(* CoDeSys 2.3.8.1 project: House.pro *)
(* Libraries: Standard.lib 4.10.05 12:14:46, IecSfc.lib 13.4.06 16:51:28, SYSLIBCALLBACK.LIB 16.4.07 17:52:46 *)

(* Global variable list: Global_Variables *)
VAR_GLOBAL
	(* Контроль 0 *)
	G_IN_CTL_BTN_1: BOOL; (* Кнопка ALL *)
	G_IN_CTL_BTN_2: BOOL; (* Кнопка RESET *)
	G_OUT_CTL_ALARM_LAMP: BOOL; (* Лампа-сигнализатор *)
	G_OUT_CTL_ALARM_SOUND: BOOL; (* Динамик в ПЛК *)
	G_OUT_CTL_SOCKET_1: BOOL := TRUE; (* Питание для МВВ *)

	(* Дверь *)
	G_IN_DOOR_DTR_1: BOOL; (* Сенсор открытия двери *)
	G_IN_DOOR_BTN_BELL: BOOL; (* Кнопка звонка *)
	G_OUT_DOOR_BELL: BOOL; (* Звонок *)

	(* Кухня 1 *)
	G_IN_KTN_BTN_1: BOOL; (* Выключатель основной *)
	G_IN_KTN_BTN_2: BOOL; (* Выключатель для вытяжки *)
	G_IN_KTN_DTR_1: BOOL; (* Датчик протечек *)
	G_OUT_KTN_LIGHT_1: BOOL; (* Свет основной *)
	G_OUT_KTN_LIGHT_2: BOOL; (* Свет второстепенный (подсветка) *)
	G_OUT_KTN_FAN_1: BOOL; (* Вытяжка *)

	(* Балкон *)
	G_IN_BLKN_BTN_1: BOOL; (* Выключатель *)
	G_OUT_BLKN_LIGHT_1: BOOL; (* Свет *)

	(* Гостиная *)
	G_IN_LVG_BTN_1: BOOL; (* Выключатель *)
	G_IN_LVG_BTN_2: BOOL; (* Выключатель на рабочем месте *)
	G_OUT_LVG_LIGHT_1: BOOL; (* Свет основной *)
	G_OUT_LVG_LIGHT_2: BOOL; (* Свет второстепенный *)

	(* Спальная *)
	G_IN_BDR_BTN_1: BOOL; (* Выключатель *)
	G_IN_BDR_BTN_2: BOOL; (* Выключатель над кроватью *)
	G_IN_BDR_BTN_3: BOOL; (* Выключатель над кроватью *)
	G_OUT_BDR_LIGHT_1: BOOL; (* Свет *)
	G_OUT_BDR_LIGHT_2: BOOL; (* Свет второстепенный *)
	G_OUT_BDR_LIGHT_3: BOOL; (* Свет над кроватью (торшер) *)
	G_OUT_BDR_LIGHT_4: BOOL; (* Свет над кроватью (торшер) *)

	(* Ванная большая *)
	G_IN_BMB_BTN_1: BOOL; (* Выключатель основной *)
	G_IN_BMB_BTN_2: BOOL; (* Выключатель около зеркала *)
	G_IN_BMB_DTR_1: BOOL; (* Датчик протечек *)
	G_OUT_BMB_LIGHT_1: BOOL; (* Свет основной *)
	G_OUT_BMB_LIGHT_2: BOOL; (* Свет около зеркала *)
	G_OUT_BMB_FAN_1: BOOL; (* Вытяжка *)
	G_OUT_BMB_VLV_1: BOOL; (* Вентиль *)
	G_OUT_BMB_VLV_2: BOOL; (* Вентиль *)

	(* Детская *)
	G_IN_CHLD_BTN_1: BOOL; (* Выключатель *)
	G_OUT_CHLD_LIGHT_1: BOOL; (* Свет основной *)
	G_OUT_CHLD_LIGHT_2: BOOL; (* Свет второстепенный *)

	(* Коридор *)
	G_IN_HLL_BTN_1: BOOL; (* Проходной выключатель *)
	G_IN_HLL_BTN_2: BOOL; (* Проходной выключатель *)
	G_IN_HLL_BTN_3: BOOL; (* Выключатель на зеркало *)
	G_IN_HLL_BTN_4: BOOL; (* Выключатель в шкафу *)
	G_IN_HLL_BTN_5: BOOL; (* Выключатель в шкафу *)

	G_OUT_HLL_LIGHT_1: BOOL; (* Свет основной *)
	G_OUT_HLL_LIGHT_2: BOOL; (* Свет второстепенный *)
	G_OUT_HLL_LIGHT_3: BOOL; (* Свет зеркало *)
	G_OUT_HLL_LIGHT_4: BOOL; (* Свет в шкафу *)
	G_OUT_HLL_LIGHT_5: BOOL; (* Свет в шкафу *)

	(* Ванная малая *)
	G_IN_BMS_BTN_1: BOOL; (* Выключатель *)
	G_IN_BMS_DTR_1: BOOL; (* Датчик протечек *)
	G_OUT_BMS_LIGHT_1: BOOL; (* Вытяжка *)
	G_OUT_BMS_FAN_1: BOOL; (* Вытяжка *)
	G_OUT_BMS_VLV_1: BOOL; (* Вентиль *)
	G_OUT_BMS_VLV_2: BOOL; (* Вентиль *)

	(* Розетки *)
	(* Кухня и балкон *)
	G_OUT_1_2_SOCKET_G1: BOOL; (* Общие *)
	G_OUT_1_2_SOCKET_G2: BOOL := TRUE; (* Неотключаемые (холодильник)*)
	G_OUT_1_2_SOCKET_G3: BOOL; (* Посудомойка *)
	G_OUT_1_2_SOCKET_G4: BOOL; (* Плита, 380В *)
	(* Гостиная и спальня *)
	G_OUT_3_4_SOCKET_G1: BOOL; (* Общие *)
	G_OUT_3_4_SOCKET_G2: BOOL; (* Неотключаемые (компьютер) *)
	(* Ванная большая *)
	G_OUT_5_SOCKET_G1: BOOL; (* Общие *)
	G_OUT_5_SOCKET_G2: BOOL := TRUE; (* Стиральная машина *)
	G_OUT_5_SOCKET_G3: BOOL; (* Резерв на бойлер и (или) баню *)
	(* Коридор и детская *)
	G_OUT_6_7_SOCKET_G1: BOOL; (* Общие *)
	G_OUT_6_7_SOCKET_G2: BOOL := TRUE; (* Неотключаемые (рядом со щитком, роутер, сервер и т.п.) *)

END_VAR

(* POU PLC_PRG, ST *)
PROGRAM PLC_PRG
VAR
	KTN_BTN_1 : Z_FB_DIFF_OUT_ON_LONG_AND_SHORT;
	KTN_BTN_2 : Z_FB_SINGLE_SW;

	BLKN_BTN : Z_FB_SINGLE_SW;

	LVG_BTN : Z_FB_SHORT_P_OUT1_LONG_P_OUT1_AND_OUT2;

	BDR_BTN_1 : Z_FB_SHORT_P_OUT1_LONG_P_OUT1_AND_OUT2;
	BDR_BTN_2 : Z_FB_SINGLE_SW;
	BDR_BTN_3 : Z_FB_SINGLE_SW;

	BMB_BTN_1 : Z_FB_SHRT_P_OUT1_LNG_P_OUT1_OUT2_TIMER;
	BMB_BTN_2 : Z_FB_SINGLE_SW;

	CHLD_BTN : Z_FB_SHORT_P_OUT1_LONG_P_OUT1_AND_OUT2;

	HLL_BTN_1_2 : FB_HLL;
	HLL_BTN_3 : Z_FB_SINGLE_SW_WITH_TIMER;
	HLL_BTN_4 : Z_FB_SINGLE_SW_WITH_TIMER;
	HLL_BTN_5 : Z_FB_SINGLE_SW_WITH_TIMER;

	BMS_BTN : Z_FB_SHRT_P_OUT1_LNG_P_OUT1_OUT2_TIMER;

	CTL_BTN_ALL : FB_ALL;

	IN_WS_LEFT : Z_FB_WS;
	IN_WS_RIGHT : Z_FB_WS;

	T_LONG_PRESS : TIME := t#1000ms;
	T_LIGHT_OFF : TIME := t#5000ms;
	T_FAN_OFF : TIME := t#5000ms;

	ALARM : FB_ALARM;

	ERROR : BOOL;

END_VAR
(* Основной выключатель на кухне *)
KTN_BTN_1 (IN := G_IN_KTN_BTN_1, Q1 := G_OUT_KTN_LIGHT_1, Q2 := G_OUT_KTN_LIGHT_2, TC := T_LONG_PRESS);

(* Второстепенный выключатель на кухне *)
KTN_BTN_2 (IN := G_IN_KTN_BTN_2, Q :=  G_OUT_KTN_FAN_1);

(* Выключатель на балконе *)
BLKN_BTN (IN := G_IN_BLKN_BTN_1, Q := G_OUT_BLKN_LIGHT_1);

(* Выключатели в гостиной *)
LVG_BTN (IN := G_IN_LVG_BTN_1 OR G_IN_LVG_BTN_2, Q1 := G_OUT_LVG_LIGHT_1, Q2 := G_OUT_LVG_LIGHT_2, TC := T_LONG_PRESS);

(* Выключатели в спальне *)
BDR_BTN_1 (IN := G_IN_BDR_BTN_1, Q1 := G_OUT_BDR_LIGHT_1, Q2 := G_OUT_BDR_LIGHT_2, TC := T_LONG_PRESS);
BDR_BTN_2 (IN := G_IN_BDR_BTN_2, Q := G_OUT_BDR_LIGHT_3);
BDR_BTN_3 (IN := G_IN_BDR_BTN_3, Q := G_OUT_BDR_LIGHT_4);

(* Выключатель в санузле *)
BMB_BTN_1 (IN := G_IN_BMB_BTN_1, Q1 := G_OUT_BMB_LIGHT_1, Q2 := G_OUT_BMB_FAN_1, TC := T_LONG_PRESS, TLight := T_LIGHT_OFF, TFan := T_FAN_OFF);
BMB_BTN_2 (IN := G_IN_BMB_BTN_2, Q := G_OUT_BMB_LIGHT_2);

(* Выключатели в детской *)
CHLD_BTN (IN := G_IN_CHLD_BTN_1, Q1 := G_OUT_CHLD_LIGHT_1, Q2 := G_OUT_CHLD_LIGHT_2, TC := T_LONG_PRESS);

(* Выключатель в коридоре *)
HLL_BTN_1_2 (IN := G_IN_HLL_BTN_1 OR G_IN_HLL_BTN_2, Q1 := G_OUT_HLL_LIGHT_1, Q2 := G_OUT_HLL_LIGHT_2, TC := T_LONG_PRESS);
HLL_BTN_3 (IN := G_IN_HLL_BTN_3, Q :=G_OUT_HLL_LIGHT_3, TC := T_LIGHT_OFF);
HLL_BTN_4 (IN := G_IN_HLL_BTN_4, Q :=G_OUT_HLL_LIGHT_4, TC := T_LIGHT_OFF);
HLL_BTN_5 (IN := G_IN_HLL_BTN_5, Q :=G_OUT_HLL_LIGHT_5, TC := T_LIGHT_OFF);

(* Выключатель в санузле *)
BMS_BTN (IN := G_IN_BMS_BTN_1, Q1 := G_OUT_BMS_LIGHT_1, Q2 := G_OUT_BMS_FAN_1, TC := T_LONG_PRESS, TLight := T_LIGHT_OFF, TFan := T_FAN_OFF);

(* Дверной звонок *)
(* TODO *)

(* Датчики протечек слева *)
IN_WS_LEFT(IN := G_IN_KTN_DTR_1 OR G_IN_BMS_DTR_1, RESET := G_IN_CTL_BTN_2, Q1 := G_OUT_BMS_VLV_1, Q2 := G_OUT_BMS_VLV_2, ALARM => ERROR);

(* Датчики протечек справа *)
IN_WS_RIGHT(IN := G_IN_BMB_DTR_1, RESET := G_IN_CTL_BTN_2, Q1 := G_OUT_BMB_VLV_1, Q2 := G_OUT_BMB_VLV_2, ALARM => ERROR);

(* Обработка тревоги *)
ALARM(ERROR := ERROR, Q1 := G_OUT_CTL_ALARM_LAMP, Q2 := G_OUT_CTL_ALARM_SOUND);

(* Общий выключатель *)
CTL_BTN_ALL(IN := G_IN_CTL_BTN_1, TC := T_LONG_PRESS);

(* Обработка общего выключателя *)
IF CTL_BTN_ALL.Q1 THEN

	G_OUT_KTN_LIGHT_1 := FALSE;
	G_OUT_KTN_LIGHT_2 := FALSE;
	G_OUT_KTN_FAN_1 := FALSE;

	G_OUT_BLKN_LIGHT_1 := FALSE;

	G_OUT_BMS_LIGHT_1 := FALSE;
	G_OUT_BMS_FAN_1 := FALSE;

ELSIF CTL_BTN_ALL.Q2 THEN

	G_OUT_1_2_SOCKET_G1 := FALSE;
	G_OUT_1_2_SOCKET_G3 := FALSE;
	G_OUT_1_2_SOCKET_G4 := FALSE;

	G_OUT_3_4_SOCKET_G1 := FALSE;
	G_OUT_3_4_SOCKET_G2 := FALSE;

	G_OUT_5_SOCKET_G1 := FALSE;
	G_OUT_5_SOCKET_G3 := FALSE;

	G_OUT_6_7_SOCKET_G1 := FALSE;

ELSE

	G_OUT_1_2_SOCKET_G1 := CTL_BTN_ALL.G1_STATE;
	G_OUT_1_2_SOCKET_G3 := CTL_BTN_ALL.G1_STATE;
	G_OUT_1_2_SOCKET_G4 := CTL_BTN_ALL.G1_STATE;

	G_OUT_3_4_SOCKET_G1 := CTL_BTN_ALL.G1_STATE;
	G_OUT_3_4_SOCKET_G2 := CTL_BTN_ALL.G1_STATE;

	G_OUT_5_SOCKET_G1 := CTL_BTN_ALL.G1_STATE;
	G_OUT_5_SOCKET_G3 := CTL_BTN_ALL.G1_STATE;

	G_OUT_6_7_SOCKET_G1 := CTL_BTN_ALL.G1_STATE;

END_IF;
END_PROGRAM

(* POU Z_FB_DIFF_OUT_ON_LONG_AND_SHORT, ST *)
(* Обработка длинного и короткого нажатия на два независимых выхода *)

FUNCTION_BLOCK Z_FB_DIFF_OUT_ON_LONG_AND_SHORT
VAR_INPUT
	IN : BOOL;
   	TC : TIME;
END_VAR
VAR_IN_OUT
	Q1 : BOOL;
	Q2 : BOOL;
END_VAR
VAR
	TX : TON;
	MEM1 : BOOL;
	MEM2 : BOOL;
END_VAR
TX(IN := IN, PT := TC);

IF TX.Q AND NOT MEM2 AND IN THEN
	Q2 := NOT Q2;
ELSIF NOT IN AND MEM1 AND NOT MEM2 THEN
	Q1 := NOT Q1;
END_IF;

MEM1 :=  IN;
MEM2 := TX.Q;
END_FUNCTION_BLOCK

(* POU Z_FB_SINGLE_SW, ST *)
(* Кнопка как выключатель *)

FUNCTION_BLOCK Z_FB_SINGLE_SW
VAR_INPUT
	IN: BOOL;
END_VAR
VAR_IN_OUT
	Q: BOOL;
END_VAR
VAR
	MEM : BOOL := FALSE;
END_VAR
IF IN AND NOT MEM THEN
	Q := NOT Q;
END_IF

MEM := IN;
END_FUNCTION_BLOCK

(* POU Z_FB_SHORT_P_OUT1_LONG_P_OUT1_AND_OUT2, ST *)
(* Два выхода
первый - короткое нажатие
первый и второй - длинное нажатие*)
FUNCTION_BLOCK Z_FB_SHORT_P_OUT1_LONG_P_OUT1_AND_OUT2
VAR_INPUT
	IN : BOOL;
   	TC : TIME;
END_VAR
VAR_IN_OUT
	Q1 : BOOL;
	Q2 : BOOL;
END_VAR
VAR
	TX : TON;
	MEM1, MEM2 : BOOL;
END_VAR
TX(IN := IN, PT := TC);

IF IN AND NOT MEM1 THEN
      Q1 := NOT Q1;
      IF NOT Q1 THEN
         Q2 := FALSE;
      END_IF
END_IF

IF TX.Q AND NOT MEM2 AND Q1 THEN
      Q2 := TRUE;
END_IF;

MEM1 := IN;
MEM2 := TX.Q;
END_FUNCTION_BLOCK

(* POU Z_FB_SHRT_P_OUT1_LNG_P_OUT1_OUT2_TIMER, ST *)
(* Два выхода
первый - короткое нажатие
первый и второй - длинное нажатие
при OUT2 = TRUE и длинном нажатии отключается OUT1 и OUT2, 
при OUT1 = TRUE и коротком нажатии отключается OUT1, а OUT2 отключается по таймеру
при OUT1 = TRUE OUT1 отключается по таймеру
*)
FUNCTION_BLOCK Z_FB_SHRT_P_OUT1_LNG_P_OUT1_OUT2_TIMER
VAR_INPUT
	IN : BOOL;
   	TC : TIME;
	TFan : TIME;
	TLight : TIME;
END_VAR
VAR_IN_OUT
	Q1 : BOOL;
	Q2 : BOOL;
END_VAR
VAR
	TX : TON;
	TPFanInst : TOF;
	TPLightInst : TP;
	MEM1, MEM2 : BOOL;
END_VAR
TX(IN := IN, PT := TC);

IF TX.Q AND NOT MEM2 AND IN THEN
	Q1 := NOT Q1;
	Q2 := NOT Q2;
ELSIF NOT IN AND MEM1 AND NOT MEM2 THEN
	Q1 := NOT Q1;
END_IF

TPFanInst(PT := TFan, IN := Q1);
IF Q2 AND NOT TPFanInst.Q THEN
	Q2 := TPFanInst.Q;
END_IF

TPLightInst(PT := TLight, IN := Q1);
IF Q1 AND NOT TPLightInst.Q THEN
	Q1 := TPLightInst.Q;
	Q2 := TPLightInst.Q;
END_IF

(*AND NOT MEM2 AND IN THEN
	Q2 := NOT Q2;
	Q1 := NOT Q1;
ELSIF NOT IN AND MEM1 THEN
	(*IF NOT MEM2 AND NOT Q2 THEN*)
		Q1 := NOT Q1;
	ELSIF NOT MEM2 AND MEM1 THEN
		Q2 := NOT Q2;
	END_IF;
END_IF;*)

MEM1 :=  IN;
MEM2 := TX.Q;
END_FUNCTION_BLOCK

(* POU FB_HLL, ST *)
FUNCTION_BLOCK FB_HLL
VAR_INPUT
	IN : BOOL;
   	TC : TIME;
END_VAR
VAR_IN_OUT
	Q1 : BOOL;
	Q2 : BOOL;
END_VAR
VAR
	TX : TON;
	MEM1, MEM2 : BOOL;
END_VAR
TX(IN := IN, PT := TC);

IF TX.Q AND NOT MEM2 AND IN THEN
	Q2 := NOT Q2;
ELSIF NOT IN AND MEM1 THEN
	IF NOT MEM2 AND NOT Q2 THEN
		Q1 := NOT Q1;
	ELSIF NOT MEM2 AND MEM1 THEN
		Q2 := NOT Q2;
	END_IF;
END_IF;

MEM1 :=  IN;
MEM2 := TX.Q;
END_FUNCTION_BLOCK

(* POU Z_FB_SINGLE_SW_WITH_TIMER, ST *)
(* Кнопка как выключатель c таймером на отключение *)
FUNCTION_BLOCK Z_FB_SINGLE_SW_WITH_TIMER
VAR_INPUT
	IN: BOOL;
	TC : TIME;
END_VAR
VAR_IN_OUT
	Q: BOOL;
END_VAR
VAR
	MEM : BOOL := FALSE;
	TPInst : TP;
END_VAR
IF IN AND NOT MEM THEN
	Q := NOT Q;
END_IF

TPInst(PT := TC, IN := Q);
IF Q AND NOT TPInst.Q THEN
	Q := TPInst.Q;
END_IF

MEM := IN;
END_FUNCTION_BLOCK

(* POU FB_ALL, ST *)
FUNCTION_BLOCK FB_ALL
VAR_INPUT
	IN: BOOL;
	TC : TIME;
END_VAR
VAR_OUTPUT
	Q1: BOOL := FALSE;
	Q2: BOOL := FALSE;
	G1_STATE: BOOL := TRUE;
END_VAR
VAR
	TX: TON;
	MEM: BOOL;
END_VAR
TX(IN := IN, PT := TC);

IF IN THEN
	IF TX.Q AND NOT MEM THEN
		Q2 := TRUE;
	ELSIF TX.Q AND MEM THEN
		G1_STATE := FALSE;
	ELSIF NOT MEM THEN
		Q1 := TRUE;
		G1_STATE := TRUE;
	END_IF;
ELSE
	Q1 := FALSE;
	Q2 := FALSE;
END_IF;

MEM := TX.Q;
END_FUNCTION_BLOCK

(* POU Z_FB_WS, ST *)
(* Слушаем сенсоры слева *)

FUNCTION_BLOCK Z_FB_WS
VAR_INPUT
	IN : BOOL;
	RESET : BOOL;
END_VAR
VAR_IN_OUT
	Q1 : BOOL;
	Q2 : BOOL;
END_VAR
VAR_OUTPUT
	ALARM : BOOL := FALSE;
END_VAR
VAR
	MEM : BOOL := FALSE;
END_VAR
IF IN THEN
	Q1 := TRUE;
	Q2 := TRUE;
	ALARM := TRUE;
ELSIF RESET THEN
	Q1 := FALSE;
	Q2 := FALSE;
	ALARM := FALSE;
END_IF

MEM := IN;
END_FUNCTION_BLOCK

(* POU FB_ALARM, ST *)
FUNCTION_BLOCK FB_ALARM
VAR_INPUT
	ERROR : BOOL;
END_VAR
VAR_IN_OUT
	Q1 : BOOL;
	Q2 : BOOL;
END_VAR
VAR
	tProcessTime : TIME;
	tmTimer : TON := (PT:= T#2s);
	Q: BOOL;
END_VAR
IF ERROR THEN
	tmTimer(IN := tProcessTime < T#2S, ET => tProcessTime);
	Q := tProcessTime < T#1S;
ELSE
	Q := FALSE;
END_IF;
Q1 := Q;
Q2 := Q;
END_FUNCTION_BLOCK
